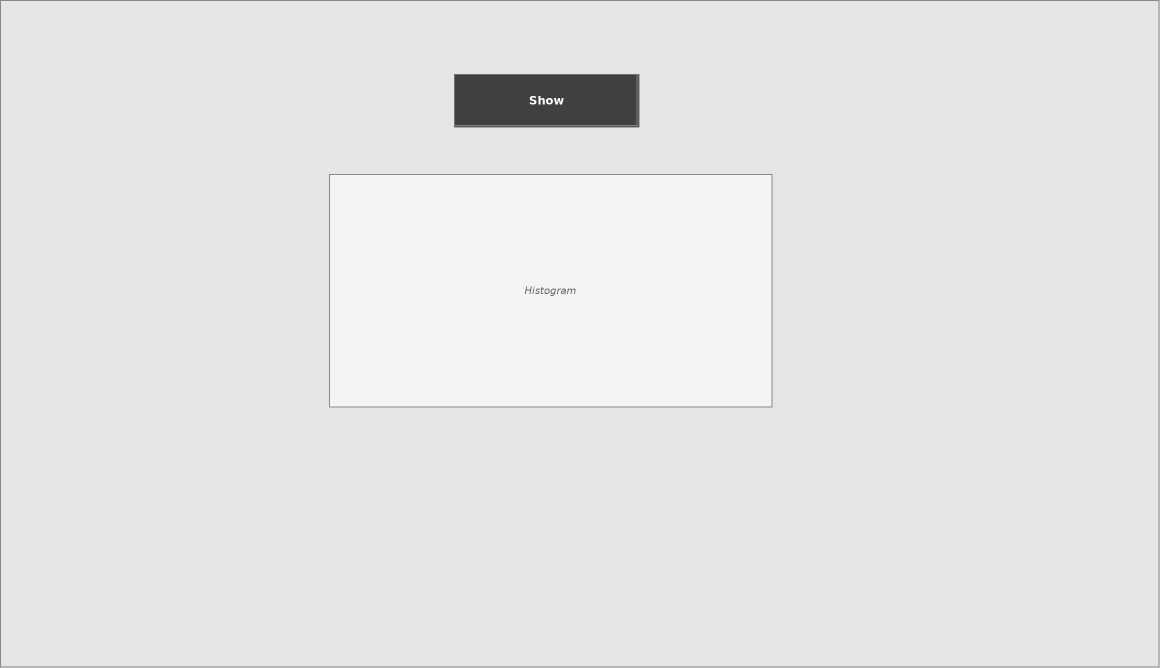
VISUALIZATION V_Trend  // 1160x668
VAR_IN_OUT
	arrHistogram 							: ARRAY [1..20] OF INT;
	bShow 									: BOOL;
END_VAR
    Histogram (329,174 443x233), scale format: %.1f, scale 0..40
        p1518820177: arrHistogram
        p102497268: arrHistogram
        p788070771: ARRAY [1..20] OF INT
    Button (454,74 185x53), "Show", colour toggle: bShow
        toggle bShow
END_VISUALIZATION

(* stored: Version 1.1.0.1, ProductVersion 3.1.4024.3
   Visu V_Trend: Id {976b530a-521a-48c9-9b88-41b61aaceff4} *)
